// Mitsubishi GX Works2 project: plc-ladder   PLC: FX3U/FX3UC

PROGRAM MAIN
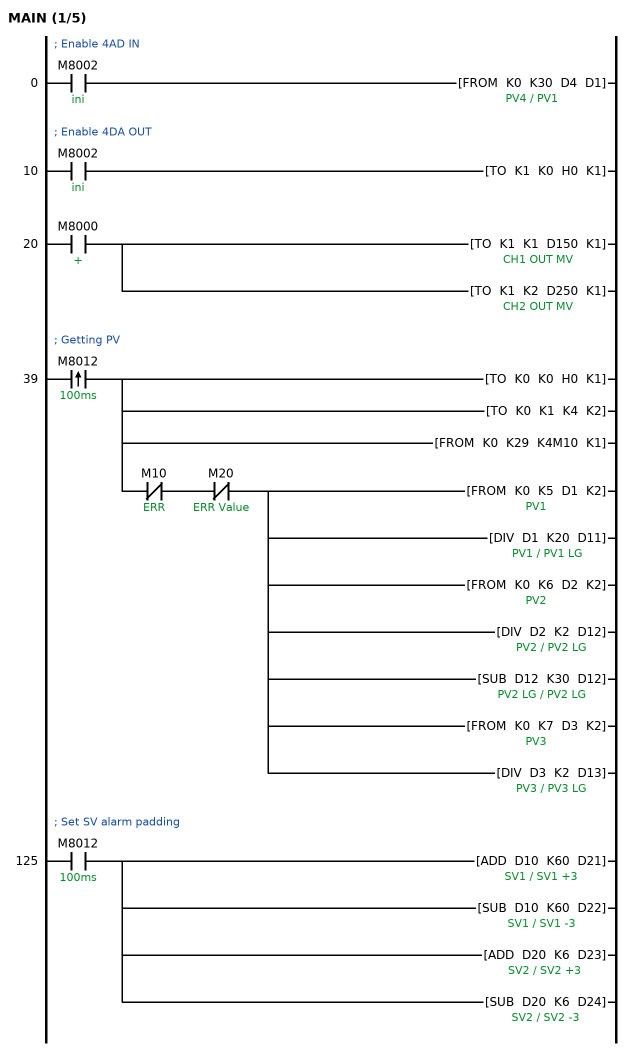
; Enable 4AD IN
0     LD      M8002  ; ini
      FROM    K0 K30 D4 D1  ; PV4 / PV1
; Enable 4DA OUT
10    LD      M8002  ; ini
      TO      K1 K0 H0 K1
20    LD      M8000  ; +
      TO      K1 K1 D150 K1  ; CH1 OUT MV
      TO      K1 K2 D250 K1  ; CH2 OUT MV
; Getting PV
39    LDP     M8012  ; 100ms
      TO      K0 K0 H0 K1
      TO      K0 K1 K4 K2
      FROM    K0 K29 K4M10 K1  ; ERR
      ANI     M10  ; ERR
      ANI     M20  ; ERR Value
      FROM    K0 K5 D1 K2
      DIV     D1 K20 D11  ; PV1 LG
      FROM    K0 K6 D2 K2  ; PV2
      DIV     D2 K2 D12  ; PV2 LG
      SUB     D12 K30 D12
      FROM    K0 K7 D3 K2  ; PV3
      DIV     D3 K2 D13  ; PV3 LG
; Set SV alarm padding
125   LD      M8012  ; 100ms
      ADD     D10 K60 D21  ; SV1 / SV1 +3
      SUB     D10 K60 D22  ; SV1 -3
      ADD     D20 K6 D23  ; SV2 / SV2 +3
      SUB     D20 K6 D24  ; SV2 -3
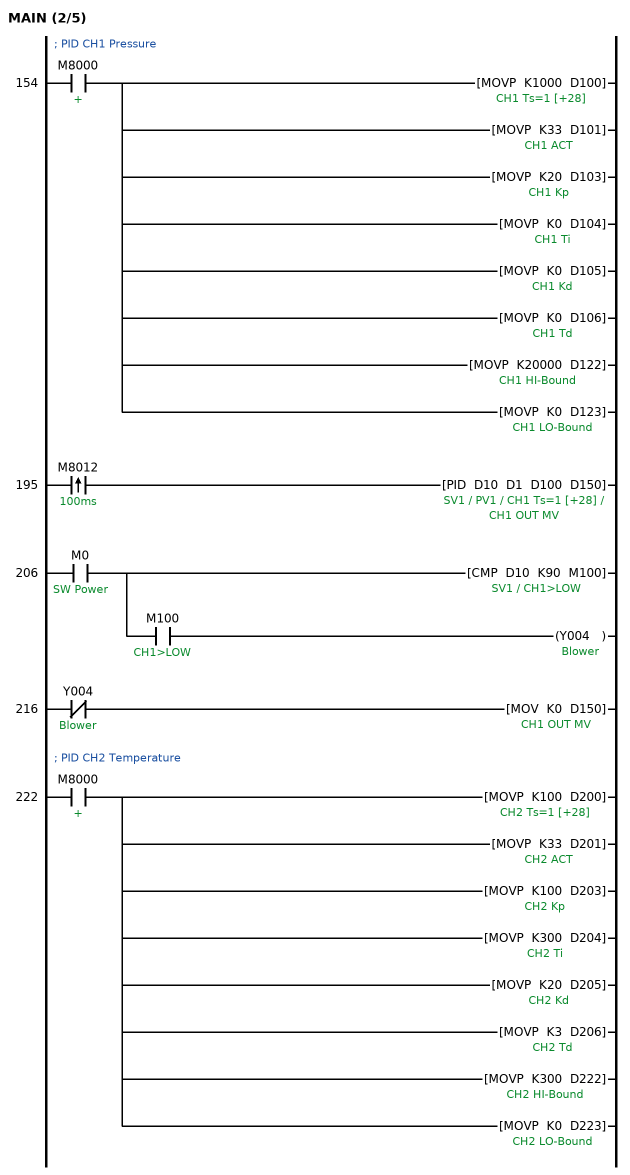
; PID CH1 Pressure
154   LD      M8000  ; +
      MOVP    K1000 D100  ; CH1 Ts=1 [+28]
      MOVP    K33 D101  ; CH1 ACT
      MOVP    K20 D103  ; CH1 Kp
      MOVP    K0 D104  ; CH1 Ti
      MOVP    K0 D105  ; CH1 Kd
      MOVP    K0 D106  ; CH1 Td
      MOVP    K20000 D122  ; CH1 HI-Bound
      MOVP    K0 D123  ; CH1 LO-Bound
195   LDP     M8012  ; 100ms
      PID     D10 D1 D100 D150
206   LD      M0  ; SW Power
      CMP     D10 K90 M100  ; CH1>LOW
      AND     M100  ; CH1>LOW
      OUT     Y004  ; Blower
216   LDI     Y004  ; Blower
      MOV     K0 D150
; PID CH2 Temperature
222   LD      M8000  ; +
      MOVP    K100 D200  ; CH2 Ts=1 [+28]
      MOVP    K33 D201  ; CH2 ACT
      MOVP    K100 D203  ; CH2 Kp
      MOVP    K300 D204  ; CH2 Ti
      MOVP    K20 D205  ; CH2 Kd
      MOVP    K3 D206  ; CH2 Td
      MOVP    K300 D222  ; CH2 HI-Bound
      MOVP    K0 D223  ; CH2 LO-Bound
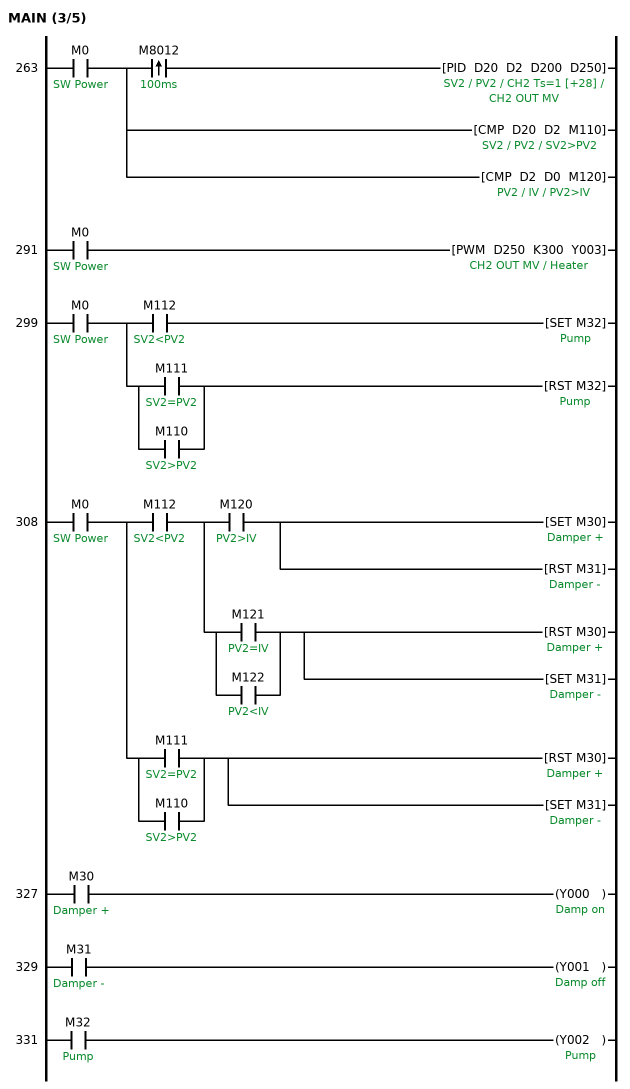
263   LD      M0  ; SW Power
      MPS
      ANDP    M8012  ; 100ms
      PID     D20 D2 D200 D250
      MPP
      CMP     D20 D2 M110  ; SV2>PV2
      CMP     D2 D0 M120  ; IV / PV2>IV
291   LD      M0  ; SW Power
      PWM     D250 K300 Y003  ; Heater
299   LD      M0  ; SW Power
      MPS
      AND     M112  ; SV2<PV2
      SET     M32  ; Pump
      MPP
      LD      M111  ; SV2=PV2
      OR      M110  ; SV2>PV2
      ANB
      RST     M32  ; Pump
308   LD      M0  ; SW Power
      MPS
      AND     M112  ; SV2<PV2
      MPS
      AND     M120  ; PV2>IV
      SET     M30  ; Damper +
      RST     M31  ; Damper -
      MPP
      LD      M121  ; PV2=IV
      OR      M122  ; PV2<IV
      ANB
      RST     M30  ; Damper +
      SET     M31  ; Damper -
      MPP
      LD      M111  ; SV2=PV2
      OR      M110  ; SV2>PV2
      ANB
      RST     M30  ; Damper +
      SET     M31  ; Damper -
327   LD      M30  ; Damper +
      OUT     Y000  ; Damp on
329   LD      M31  ; Damper -
      OUT     Y001  ; Damp off
331   LD      M32  ; Pump
      OUT     Y002  ; Pump
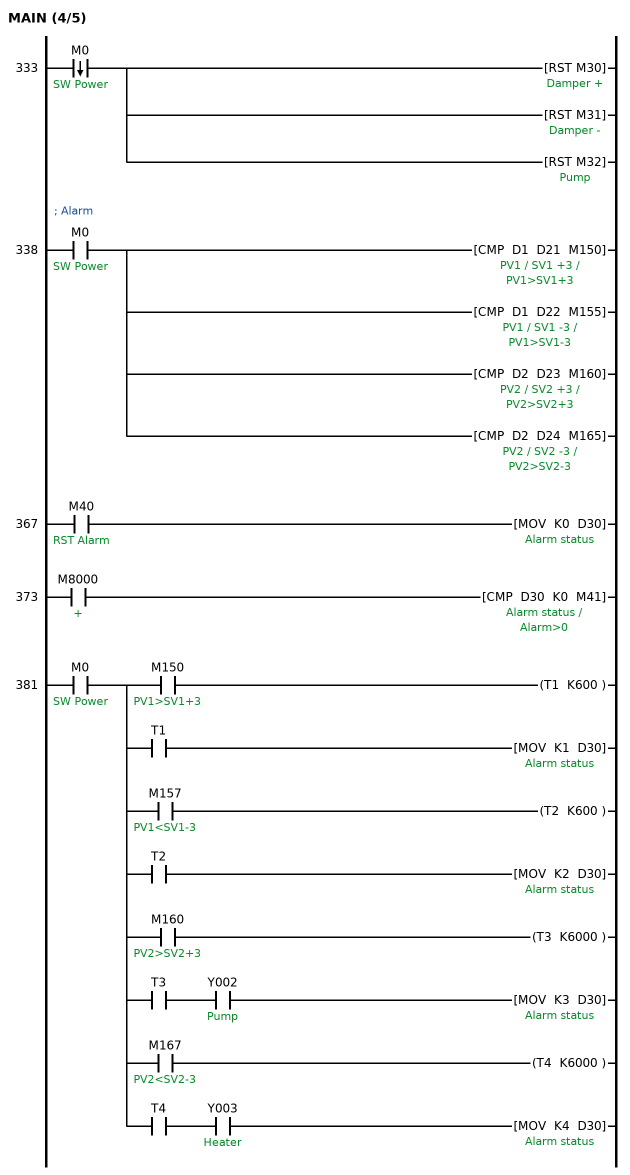
333   LDF     M0  ; SW Power
      RST     M30  ; Damper +
      RST     M31  ; Damper -
      RST     M32  ; Pump
; Alarm
338   LD      M0  ; SW Power
      CMP     D1 D21 M150  ; PV1>SV1+3
      CMP     D1 D22 M155  ; PV1>SV1-3
      CMP     D2 D23 M160  ; PV2>SV2+3
      CMP     D2 D24 M165  ; PV2>SV2-3
367   LD      M40  ; RST Alarm
      MOV     K0 D30  ; Alarm status
373   LD      M8000  ; +
      CMP     D30 K0 M41  ; Alarm>0
381   LD      M0  ; SW Power
      MPS
      AND     M150  ; PV1>SV1+3
      OUT     T1 K600
      MRD
      AND     T1
      MOV     K1 D30
      MRD
      AND     M157  ; PV1<SV1-3
      OUT     T2 K600
      MRD
      AND     T2
      MOV     K2 D30
      MRD
      AND     M160  ; PV2>SV2+3
      OUT     T3 K6000
      MRD
      AND     T3
      AND     Y002  ; Pump
      MOV     K3 D30
      MRD
      AND     M167  ; PV2<SV2-3
      OUT     T4 K6000
      MPP
      AND     T4
      AND     Y003  ; Heater
      MOV     K4 D30
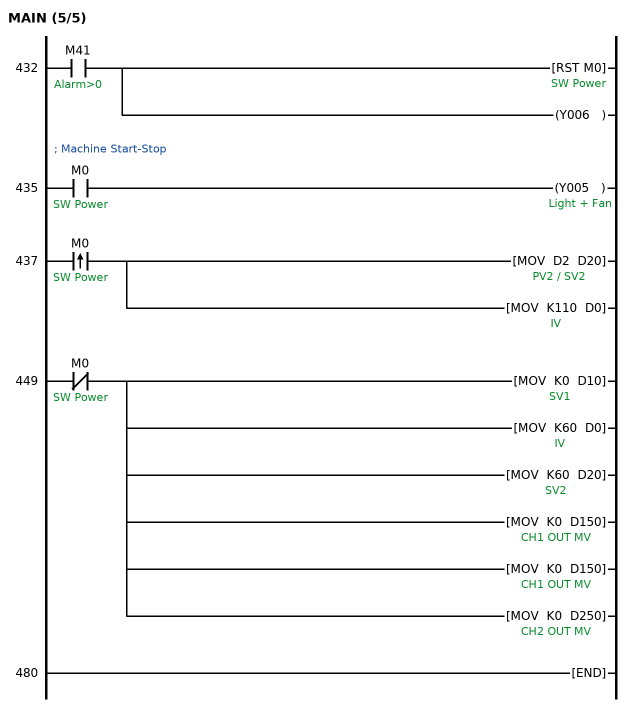
432   LD      M41  ; Alarm>0
      RST     M0  ; SW Power
      OUT     Y006
; Machine Start-Stop
435   LD      M0  ; SW Power
      OUT     Y005  ; Light + Fan
437   LDP     M0  ; SW Power
      MOV     D2 D20
      MOV     K110 D0
449   LDI     M0  ; SW Power
      MOV     K0 D10
      MOV     K60 D0
      MOV     K60 D20
      MOV     K0 D150
      MOV     K0 D150
      MOV     K0 D250
480   END
END_PROGRAM

// device comments not shown above
M42  ; Alarm=0
M43  ; Alarm<0
M101  ; CH1=LOW
M102  ; CH1<LOW
M151  ; PV1=SV1+3
M152  ; PV1<SV1+3
M156  ; PV1=SV1-3
M161  ; PV2=SV2+3
M162  ; PV2<SV2+3
M166  ; PV2=SV2-3
M555  ; comment
M1000  ; Test On-Off
M2000  ; Comment Off
